DATA_BLOCK "KeyenceSR1000Ctrl_803A1DB"
{ S7_Optimized_Access := 'FALSE' }
VERSION : 0.1
NON_RETAIN
// ATTRIBUTES
// AUTO_NUMBER = False
// BLOCK_NUMBER = 1802
// END_ATTRIBUTES
"KeyenceSR1000Ctrl"

BEGIN

END_DATA_BLOCK

